// TwinCAT 3 PLC project PLC1
// ProgramVersion: 3.1.4024.0
// libraries:
//   Tc2_Standard, * (Beckhoff Automation GmbH)
//   Tc2_System, * (Beckhoff Automation GmbH)
//   Tc3_Module, * (Beckhoff Automation GmbH)
// project tree:
//   GVLs/ GVL.TcGVL
//   / PlcTask.TcTTO
//   POUs/ FB_Clock.TcPOU, MAIN.TcPOU

CONFIGURATION PLC1
    RESOURCE PLC ON TwinCAT3
        TASK PlcTask(INTERVAL := T#10ms, PRIORITY := 20);
        PROGRAM MAIN WITH PlcTask : MAIN;
    END_RESOURCE
END_CONFIGURATION

// ---- GVLs/GVL.TcGVL
{attribute 'qualified_only'}
VAR_GLOBAL
	bClock : BOOL;
END_VAR

// ---- POUs/MAIN.TcPOU
PROGRAM MAIN
VAR
	fbClk: FB_Clock;
END_VAR

fbClk(TIME_ON:= T#10MS, TIME_OFF:= T#200MS, OUT_CLK=> GVL.bClock);

END_PROGRAM

// ---- POUs/FB_Clock.TcPOU
FUNCTION_BLOCK FB_Clock
VAR_INPUT
	TIME_ON		: TIME;	// Time to mantain clk ON
	TIME_OFF 	: TIME; // Time to mantain clk OFF
END_VAR
VAR_OUTPUT
	OUT_CLK		: BOOL; // CLK out
END_VAR
VAR
	TON_1		: TON;
	TON_2		: TON;
END_VAR

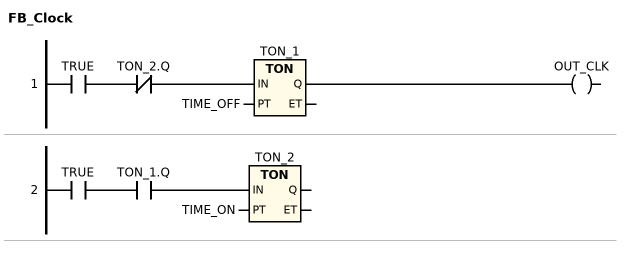
// NETWORK 1
TON_1(IN := TRUE AND NOT TON_2.Q, PT := TIME_OFF); // TON
OUT_CLK := TON_1.Q;

// NETWORK 2
TON_2(IN := TRUE AND TON_1.Q, PT := TIME_ON); // TON

END_FUNCTION_BLOCK
